PROGRAM progHSVCntrl
VAR
	HSV_04_0100 : fbHSV;

	HSV_04_1001 : fbHSV;
	HSV_04_1002 : fbHSV;
	HSV_04_1003 : fbHSV;
	HSV_04_1004 : fbHSV;
	HSV_04_1005 : fbHSV;
END_VAR

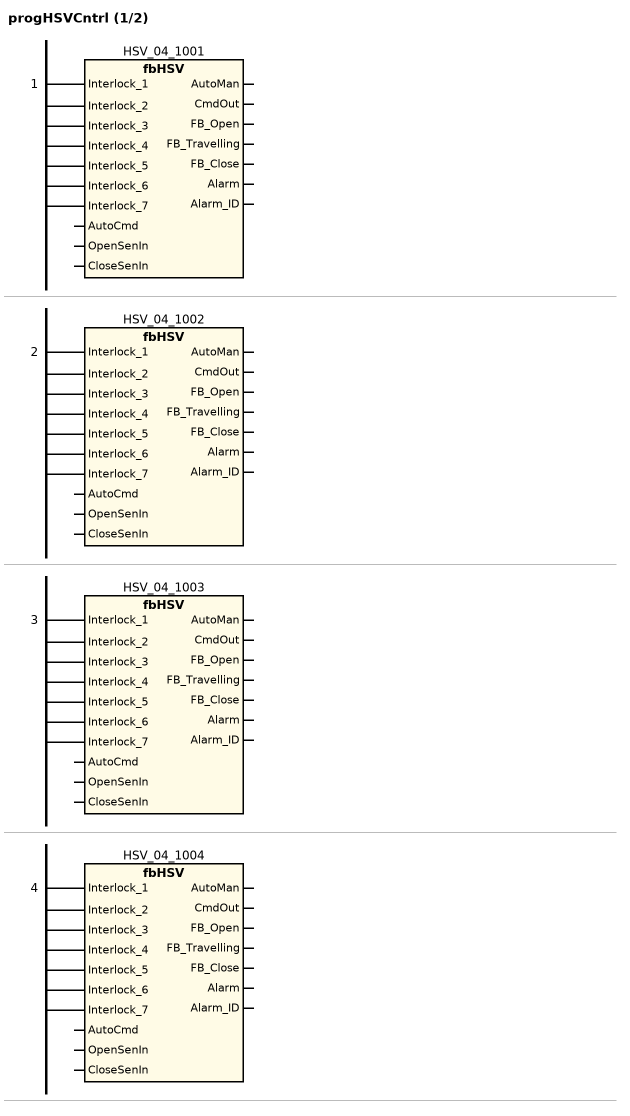
// NETWORK 1
HSV_04_1001(
    Interlock_1 := TRUE,
    Interlock_2 := TRUE,
    Interlock_3 := TRUE,
    Interlock_4 := TRUE,
    Interlock_5 := TRUE,
    Interlock_6 := TRUE,
    Interlock_7 := TRUE); // fbHSV

// NETWORK 2
HSV_04_1002(
    Interlock_1 := TRUE,
    Interlock_2 := TRUE,
    Interlock_3 := TRUE,
    Interlock_4 := TRUE,
    Interlock_5 := TRUE,
    Interlock_6 := TRUE,
    Interlock_7 := TRUE); // fbHSV

// NETWORK 3
HSV_04_1003(
    Interlock_1 := TRUE,
    Interlock_2 := TRUE,
    Interlock_3 := TRUE,
    Interlock_4 := TRUE,
    Interlock_5 := TRUE,
    Interlock_6 := TRUE,
    Interlock_7 := TRUE); // fbHSV

// NETWORK 4
HSV_04_1004(
    Interlock_1 := TRUE,
    Interlock_2 := TRUE,
    Interlock_3 := TRUE,
    Interlock_4 := TRUE,
    Interlock_5 := TRUE,
    Interlock_6 := TRUE,
    Interlock_7 := TRUE); // fbHSV

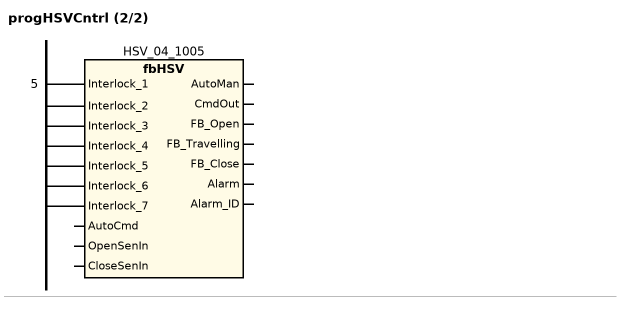
// NETWORK 5
HSV_04_1005(
    Interlock_1 := TRUE,
    Interlock_2 := TRUE,
    Interlock_3 := TRUE,
    Interlock_4 := TRUE,
    Interlock_5 := TRUE,
    Interlock_6 := TRUE,
    Interlock_7 := TRUE); // fbHSV

END_PROGRAM

(* stored: Version 1.1.0.1, ProductVersion 3.1.4022.17
   POU progHSVCntrl: Id {a7024c1e-f61a-4807-ae31-4a8a61a63135}, SpecialFunc None *)
